FUNCTION TryConvert_LREAL_TO_UINT : BOOL
VAR_INPUT
	in : LREAL;
	out : REFERENCE TO UINT;
END_VAR

IF in > DatatypeLimits.MAX_VALUE_OF_LREAL_WHICH_CAN_BE_HELD_IN_A_UINT THEN
	RETURN;
END_IF

IF in < DatatypeLimits.MIN_VALUE_OF_LREAL_WHICH_CAN_BE_HELD_IN_A_UINT THEN
	RETURN;
END_IF

out := LREAL_TO_UINT(in);
TryConvert_LREAL_TO_UINT := TRUE;

END_FUNCTION

(* stored: Version 1.1.0.1, ProductVersion 3.1.4024.12
   POU TryConvert_LREAL_TO_UINT: Id {563be11f-2cd8-4eae-9949-5223f2a78933}, SpecialFunc None *)
